Sulje kaikki portit ... JA tarkista Steppiä seuraavassa transitioehdossa, että kaikki portit ovat kiinni
Close all gates.... and check in following transition that ALL gates are closed*)

;
END_ACTION

ACTION ResetSFC_action:
(*Reset SFC*)
SFCReset:=TRUE;
END_ACTION
END_PROGRAM

(* POU OLD/PRG_ToColourSensor, SFC *)
PROGRAM PRG_ToColourSensor
VAR_INPUT
	bReset		: BOOL;	(*Reset program*)
	bExecute		: BOOL;	(*enable and run*)
END_VAR
VAR_OUTPUT
	bDone			: BOOL;
END_VAR
VAR

	tonMoveDelay	: TON;
	SFCReset		: BOOL;
	tMoveDelay	: TIME := T#4s;
END_VAR
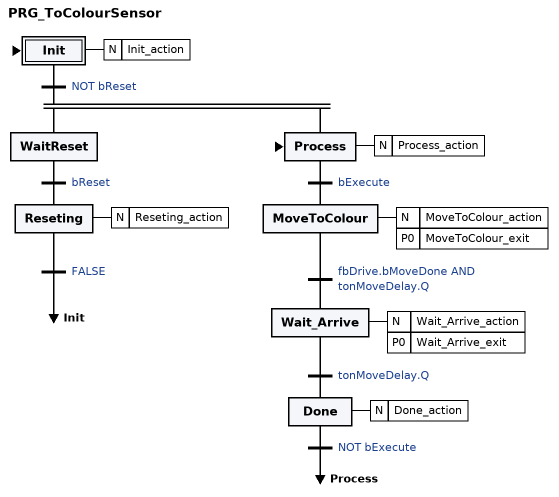
INITIAL_STEP Init:
	Init_action(N);
END_STEP
TRANSITION FROM Init TO (WaitReset, Process) := NOT bReset;
END_TRANSITION
STEP WaitReset:
END_STEP
TRANSITION FROM WaitReset TO Reseting := bReset;
END_TRANSITION
STEP Process:
	Process_action(N);
END_STEP
TRANSITION FROM Process TO MoveToColour := bExecute;
END_TRANSITION
STEP MoveToColour:
	MoveToColour_action(N);
	MoveToColour_exit(P0);
END_STEP
TRANSITION FROM MoveToColour TO Wait_Arrive := fbDrive.bMoveDone AND tonMoveDelay.Q;
END_TRANSITION
STEP Wait_Arrive:
	Wait_Arrive_action(N);
	Wait_Arrive_exit(P0);
END_STEP
TRANSITION FROM Wait_Arrive TO Done := tonMoveDelay.Q;
END_TRANSITION
STEP Done:
	Done_action(N);
END_STEP
TRANSITION FROM Done TO Process := NOT bExecute;
END_TRANSITION
STEP Reseting:
	Reseting_action(N);
END_STEP
TRANSITION FROM Reseting TO Init := FALSE;
END_TRANSITION

ACTION Init_action:
SFCReset := FALSE;
bDone := FALSE;
END_ACTION

ACTION Process_action:
bDone := FALSE;
END_ACTION

ACTION MoveToColour_action:
bDone := FALSE;

fbDrive(
	bEnable:= TRUE,
	bStart:= TRUE,
	wTarget:= GPOS_COLOR_SEN);

tonMoveDelay(IN:=TRUE , PT:= tMoveDelay);

(*
tonMoveDelay(IN:=TRUE , PT:= tMoveDelay);
*)
END_ACTION

ACTION MoveToColour_exit:
fbDrive(
	bStart:= FALSE);

tonMoveDelay(IN:=FALSE);
END_ACTION

ACTION Wait_Arrive_action:
tonMoveDelay(IN:=TRUE , PT:= tMoveDelay);
END_ACTION

ACTION Wait_Arrive_exit:
tonMoveDelay(IN:=FALSE);
END_ACTION

ACTION Done_action:
bDone := TRUE;
END_ACTION

ACTION Reseting_action:
SFCReset := TRUE;
END_ACTION
END_PROGRAM

(* POU OLD/PRG_ToColourSensor2, SFC *)
PROGRAM PRG_ToColourSensor2
VAR_INPUT
	bExecute: BOOL;
END_VAR
VAR_INPUT
	bDone: BOOL;
END_VAR
VAR
	tonMoveDelay	: TON;
	tonEjectDelay	: TON;
	tMoveDelay	: TIME := T#3s;
	tEjectorDelay	: TIME := T#3s;
END_VAR
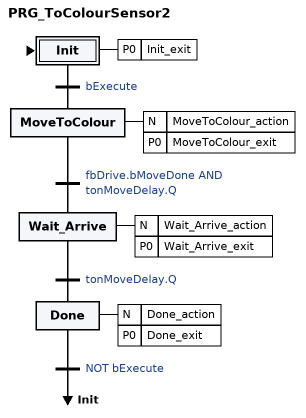
INITIAL_STEP Init:
	Init_exit(P0);
END_STEP
TRANSITION FROM Init TO MoveToColour := bExecute;
END_TRANSITION
STEP MoveToColour:
	MoveToColour_action(N);
	MoveToColour_exit(P0);
END_STEP
TRANSITION FROM MoveToColour TO Wait_Arrive := fbDrive.bMoveDone AND tonMoveDelay.Q;
END_TRANSITION
STEP Wait_Arrive:
	Wait_Arrive_action(N);
	Wait_Arrive_exit(P0);
END_STEP
TRANSITION FROM Wait_Arrive TO Done := tonMoveDelay.Q;
END_TRANSITION
STEP Done:
	Done_action(N);
	Done_exit(P0);
END_STEP
TRANSITION FROM Done TO Init := NOT bExecute;
END_TRANSITION

ACTION Init_exit:
bDone := FALSE;
END_ACTION

ACTION MoveToColour_action:
fbDrive(
	bEnable:= TRUE,
	bStart:= TRUE,
	wTarget:= GPOS_COLOR_SEN);

tonMoveDelay(IN:=TRUE , PT:= tMoveDelay);
END_ACTION

ACTION MoveToColour_exit:
fbDrive(
	bStart:= FALSE);
tonMoveDelay(IN:=FALSE);
END_ACTION

ACTION Wait_Arrive_action:
tonMoveDelay(IN:=TRUE , PT:= tMoveDelay);
END_ACTION

ACTION Wait_Arrive_exit:
tonMoveDelay(IN:=FALSE);
END_ACTION

ACTION Done_action:
bDone := TRUE;
END_ACTION

ACTION Done_exit:
bDone := FALSE;
END_ACTION
END_PROGRAM

(* POU OLD/FB_Lift2Old, SFC *)
FUNCTION_BLOCK FB_Lift2Old
VAR_INPUT
	bReset			 : BOOL;	(*Reset Request*)
	bEnable			 : BOOL;
	I_LimitUp 			 : BOOL;
	I_LimitLow 	        : BOOL;
	I_WaitingBallMetal : BOOL;

	(* ColourSensor *)
	I_SenColourYellow		:BOOL;	(*Colour sensor In1 - Yellow*)
	I_SenColourBlue		:BOOL;	(*Colour sensor In2 - Blue*)
	I_SenColourGreen		:BOOL;	(*Colour sensor In3 - Green*)
	I_SenColourRed		:BOOL;	(*Colour sensor In4 - Red*)

	(*SMEMA Handshake Inputs*)
	hiRdyToReceive_FromDS	: BOOL;
	hiBallAvail_FromUS		: BOOL;
END_VAR
VAR_OUTPUT
	bStopOK		: BOOL;
	bBallLoaded	: BOOL;
	bCurBallMetal	: BOOL;
	bCurrentBall 	: E_BallColour := NoColour;

	O_Ejector		:BOOL;

	(*SMEMA Handshake Outputs*)
	hoBallAvail_ToDS 			: BOOL;
	hoReadyToRecieve_ToUS		: BOOL;
END_VAR
VAR
	bBallRequested : BOOL := FALSE;
	fbTransferBall	:FB_TransferBall2;

	fbDelay		: FB_Wait;
	tonMoveDelay	: TON;
	tonSensorDelay	: TON;
	tTransferDelay: TIME := T#4s;
	tMoveDelay	: TIME := T#4s;
	tSensorDelay	: TIME := T#2s;
	bLocalReset	: BOOL;	(*Performs local reset*)
	SFCReset 	: BOOL;	(*Resets the execution of SFC to init once this SFCFlag is set true *)
END_VAR
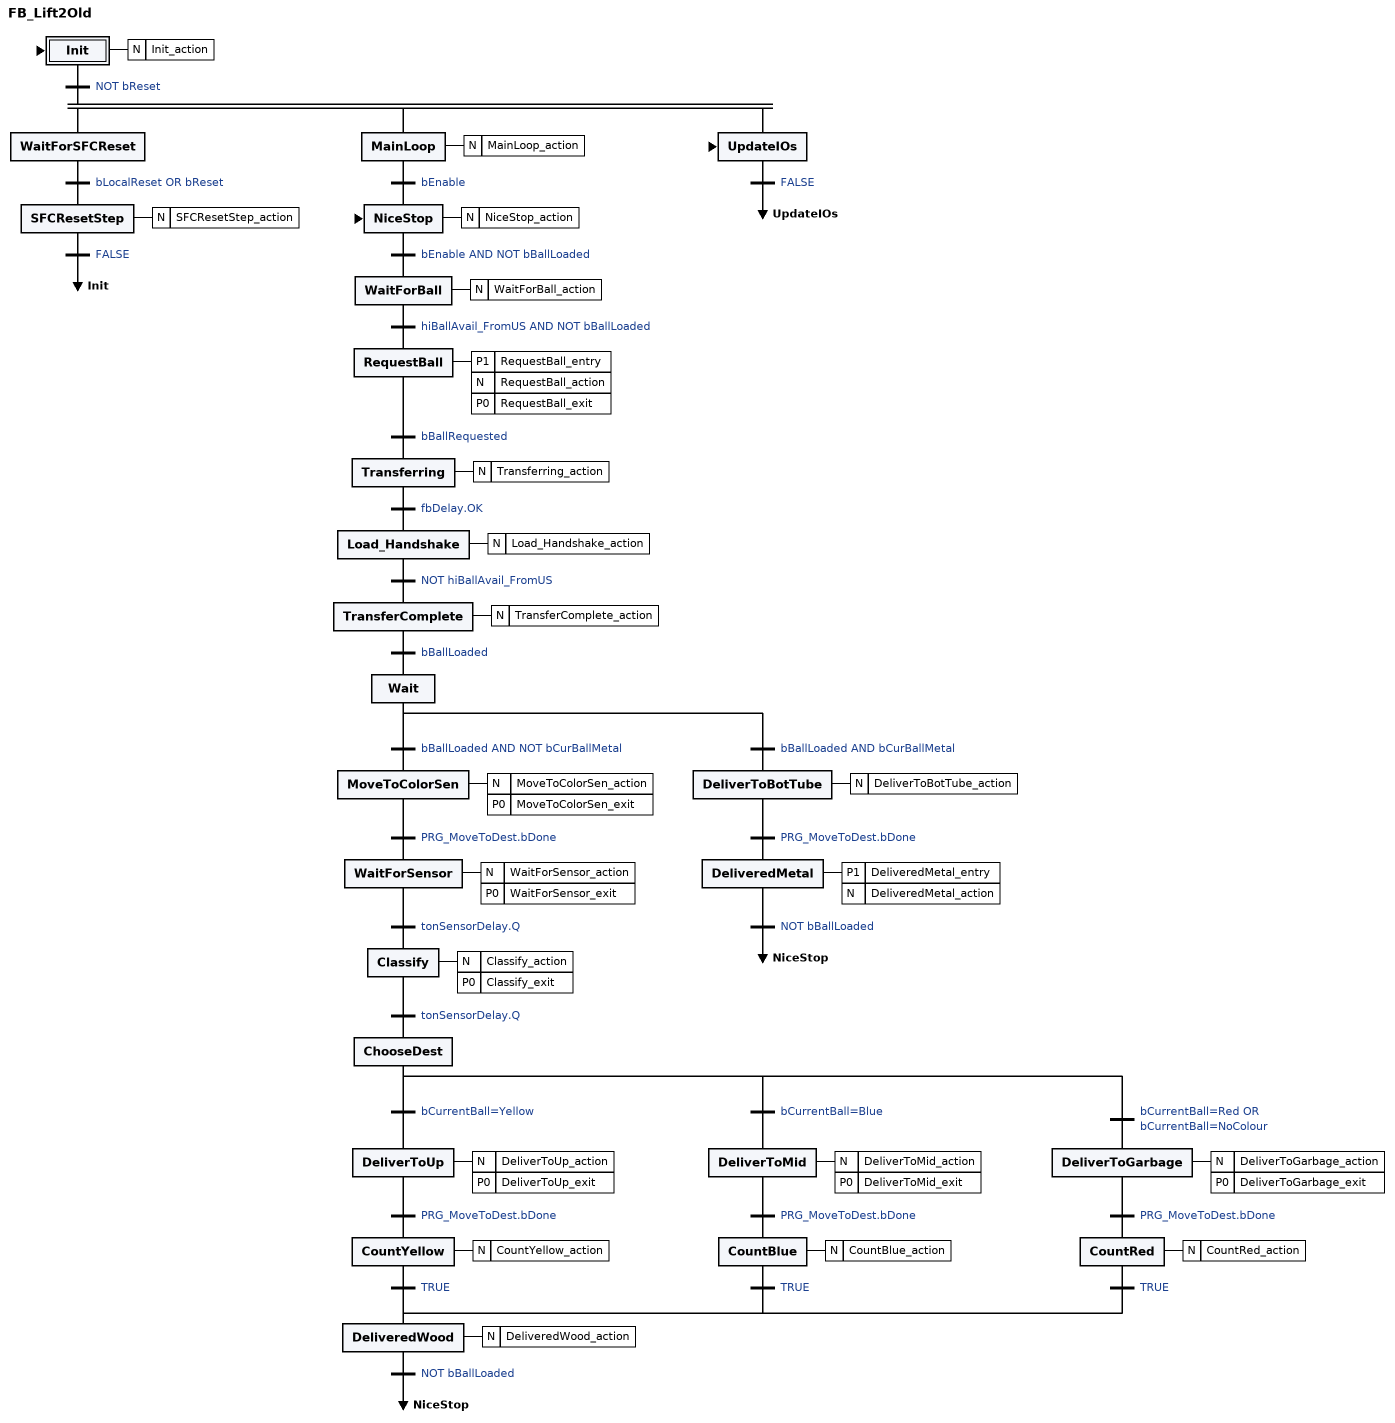
INITIAL_STEP Init:
	Init_action(N);
END_STEP
TRANSITION FROM Init TO (WaitForSFCReset, MainLoop, UpdateIOs) := NOT bReset;
END_TRANSITION
STEP WaitForSFCReset:
END_STEP
TRANSITION FROM WaitForSFCReset TO SFCResetStep := bLocalReset OR bReset;
END_TRANSITION
STEP MainLoop:
	MainLoop_action(N);
END_STEP
TRANSITION FROM MainLoop TO NiceStop := bEnable;
END_TRANSITION
STEP NiceStop:
	NiceStop_action(N);
END_STEP
TRANSITION FROM NiceStop TO WaitForBall := bEnable AND NOT bBallLoaded;
END_TRANSITION
STEP WaitForBall:
	WaitForBall_action(N);
END_STEP
TRANSITION FROM WaitForBall TO RequestBall := hiBallAvail_FromUS AND NOT bBallLoaded;
END_TRANSITION
STEP RequestBall:
	RequestBall_entry(P1);
	RequestBall_action(N);
	RequestBall_exit(P0);
END_STEP
TRANSITION FROM RequestBall TO Transferring := bBallRequested;
END_TRANSITION
STEP Transferring:
	Transferring_action(N);
END_STEP
TRANSITION FROM Transferring TO Load_Handshake := fbDelay.OK;
END_TRANSITION
STEP Load_Handshake:
	Load_Handshake_action(N);
END_STEP
TRANSITION FROM Load_Handshake TO TransferComplete := NOT hiBallAvail_FromUS;
END_TRANSITION
STEP TransferComplete:
	TransferComplete_action(N);
END_STEP
TRANSITION FROM TransferComplete TO Wait := bBallLoaded;
END_TRANSITION
STEP Wait:
END_STEP
TRANSITION FROM Wait TO MoveToColorSen := bBallLoaded AND NOT bCurBallMetal;
END_TRANSITION
TRANSITION FROM Wait TO DeliverToBotTube := bBallLoaded AND bCurBallMetal;
END_TRANSITION
STEP DeliverToBotTube:
	DeliverToBotTube_action(N);
END_STEP
TRANSITION FROM DeliverToBotTube TO DeliveredMetal := PRG_MoveToDest.bDone;
END_TRANSITION
STEP DeliveredMetal:
	DeliveredMetal_entry(P1);
	DeliveredMetal_action(N);
END_STEP
TRANSITION FROM DeliveredMetal TO NiceStop := NOT bBallLoaded;
END_TRANSITION
STEP MoveToColorSen:
	MoveToColorSen_action(N);
	MoveToColorSen_exit(P0);
END_STEP
TRANSITION FROM MoveToColorSen TO WaitForSensor := PRG_MoveToDest.bDone;
END_TRANSITION
STEP WaitForSensor:
	WaitForSensor_action(N);
	WaitForSensor_exit(P0);
END_STEP
TRANSITION FROM WaitForSensor TO Classify := tonSensorDelay.Q;
END_TRANSITION
STEP Classify:
	Classify_action(N);
	Classify_exit(P0);
END_STEP
TRANSITION FROM Classify TO ChooseDest := tonSensorDelay.Q;
END_TRANSITION
STEP ChooseDest:
END_STEP
TRANSITION FROM ChooseDest TO DeliverToUp := bCurrentBall=Yellow;
END_TRANSITION
TRANSITION FROM ChooseDest TO DeliverToMid := bCurrentBall=Blue;
END_TRANSITION
TRANSITION FROM ChooseDest TO DeliverToGarbage := bCurrentBall=Red OR bCurrentBall=NoColour;
END_TRANSITION
STEP DeliverToUp:
	DeliverToUp_action(N);
	DeliverToUp_exit(P0);
END_STEP
TRANSITION FROM DeliverToUp TO CountYellow := PRG_MoveToDest.bDone;
END_TRANSITION
STEP CountYellow:
	CountYellow_action(N);
END_STEP
TRANSITION FROM CountYellow TO DeliveredWood := TRUE;
END_TRANSITION
STEP DeliverToMid:
	DeliverToMid_action(N);
	DeliverToMid_exit(P0);
END_STEP
TRANSITION FROM DeliverToMid TO CountBlue := PRG_MoveToDest.bDone;
END_TRANSITION
STEP CountBlue:
	CountBlue_action(N);
END_STEP
TRANSITION FROM CountBlue TO DeliveredWood := TRUE;
END_TRANSITION
STEP DeliverToGarbage:
	DeliverToGarbage_action(N);
	DeliverToGarbage_exit(P0);
END_STEP
TRANSITION FROM DeliverToGarbage TO CountRed := PRG_MoveToDest.bDone;
END_TRANSITION
STEP CountRed:
	CountRed_action(N);
END_STEP
TRANSITION FROM CountRed TO DeliveredWood := TRUE;
END_TRANSITION
STEP DeliveredWood:
	DeliveredWood_action(N);
END_STEP
TRANSITION FROM DeliveredWood TO NiceStop := NOT bBallLoaded;
END_TRANSITION
STEP UpdateIOs:
END_STEP
TRANSITION FROM UpdateIOs TO UpdateIOs := FALSE;
END_TRANSITION
STEP SFCResetStep:
	SFCResetStep_action(N);
END_STEP
TRANSITION FROM SFCResetStep TO Init := FALSE;
END_TRANSITION

ACTION Init_action:
SFCReset := FALSE;
bLocalReset	:= FALSE;
END_ACTION

ACTION MainLoop_action:
hoBallAvail_ToDS			  := FALSE;
hoReadyToRecieve_ToUS := FALSE;
END_ACTION

ACTION NiceStop_action:
bStopOK	  	:= TRUE;
bCurrentBall	:= NoColour;
END_ACTION

ACTION WaitForBall_action:
bBallLoaded := FALSE;
hoReadyToRecieve_ToUS := TRUE;
END_ACTION

ACTION RequestBall_entry:
bStopOK := FALSE;
END_ACTION

ACTION RequestBall_action:
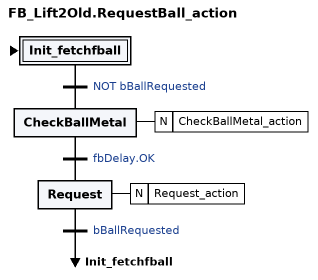
INITIAL_STEP Init_fetchfball:
END_STEP
TRANSITION FROM Init_fetchfball TO CheckBallMetal := NOT bBallRequested;
END_TRANSITION
STEP CheckBallMetal:
	CheckBallMetal_action(N);
END_STEP
TRANSITION FROM CheckBallMetal TO Request := fbDelay.OK;
END_TRANSITION
STEP Request:
	Request_action(N);
END_STEP
TRANSITION FROM Request TO Init_fetchfball := bBallRequested;
END_TRANSITION

ACTION CheckBallMetal_action:
bCurBallMetal	 := I_WaitingBallMetal;
fbDelay(IN_TIME:=T#2s);
END_ACTION

ACTION Request_action:
hoReadyToRecieve_ToUS := TRUE;
bBallRequested := TRUE;
END_ACTION
END_ACTION

ACTION RequestBall_exit:
bBallRequested := FALSE;
END_ACTION

ACTION Transferring_action:
fbDelay(IN_TIME:=tTransferDelay);
END_ACTION

ACTION Load_Handshake_action:
hoReadyToRecieve_ToUS := FALSE;
END_ACTION

ACTION TransferComplete_action:
bBallLoaded := TRUE;
END_ACTION

ACTION DeliverToBotTube_action:
PRG_MoveToDest(bExecute:= TRUE, wTarget:= GPOS_PIPE_LOW, bDone:= );
END_ACTION

ACTION DeliveredMetal_entry:
bBallLoaded := FALSE;
PRG_MoveToDest( bExecute:=FALSE);
END_ACTION

ACTION DeliveredMetal_action:
bBallLoaded := FALSE;
CountBallsSortedMetal := CountBallsSortedMetal + 1;
arrCountBallsOnTubes[1] := arrCountBallsOnTubes[1] + 1;
END_ACTION

ACTION MoveToColorSen_action:
PRG_MoveToDest(bExecute:= TRUE, wTarget:= GPOS_COLOR_SEN, bDone:= );
END_ACTION

ACTION MoveToColorSen_exit:
PRG_MoveToDest( bExecute:=FALSE);
END_ACTION

ACTION WaitForSensor_action:
tonSensorDelay(IN:=TRUE , PT:= tSensorDelay);
END_ACTION

ACTION WaitForSensor_exit:
tonSensorDelay(IN:=FALSE);
END_ACTION

ACTION Classify_action:
tonSensorDelay(IN:=TRUE , PT:= tSensorDelay);
IF I_SenColourYellow THEN
	bCurrentBall := Yellow;
ELSIF  I_SenColourBlue THEN
	bCurrentBall := Blue;
ELSIF  I_SenColourRed THEN
	bCurrentBall := Red;
ELSE
	bCurrentBall := NoColour;
END_IF
END_ACTION

ACTION Classify_exit:
tonSensorDelay(IN:=FALSE);
END_ACTION

ACTION DeliverToUp_action:
PRG_MoveToDest(bExecute:= TRUE , wTarget:= GPOS_PIPE_UP, bDone:= );
END_ACTION

ACTION DeliverToUp_exit:
PRG_MoveToDest(bExecute:= FALSE);
END_ACTION

ACTION CountYellow_action:
CountBallsSortedYellow := CountBallsSortedYellow + 1;
CountBallsSortedWooden := CountBallsSortedWooden + 1;
arrCountBallsOnTubes[3] := arrCountBallsOnTubes[3] + 1;
END_ACTION

ACTION DeliverToMid_action:
PRG_MoveToDest(bExecute:= TRUE , wTarget:= GPOS_PIPE_MID, bDone:= );
END_ACTION

ACTION DeliverToMid_exit:
PRG_MoveToDest(bExecute:= FALSE);
END_ACTION

ACTION CountBlue_action:
CountBallsSortedBlue := CountBallsSortedBlue + 1;
CountBallsSortedWooden := CountBallsSortedWooden + 1;
arrCountBallsOnTubes[2] := arrCountBallsOnTubes[2] + 1;
END_ACTION

ACTION DeliverToGarbage_action:
PRG_MoveToDest(bExecute:= TRUE , wTarget:= GPOS_GARBAGE, bDone:= );
END_ACTION

ACTION DeliverToGarbage_exit:
PRG_MoveToDest(bExecute:= FALSE);
END_ACTION

ACTION CountRed_action:
CountBallsSortedRed := CountBallsSortedRed + 1;
CountBallsSortedGarbage := CountBallsSortedGarbage + 1;
CountBallsSortedWooden := CountBallsSortedWooden + 1;
arrCountBallsOnTubes[4] := arrCountBallsOnTubes[4] + 1;
END_ACTION

ACTION DeliveredWood_action:
bBallLoaded := FALSE;
bCurrentBall := NoColour;
END_ACTION

ACTION SFCResetStep_action:
SFCReset := TRUE;
END_ACTION
END_FUNCTION_BLOCK

(* POU OLD/FB_TransferBall2, ST *)
FUNCTION_BLOCK FB_TransferBall2
VAR_INPUT
	bExecute			: BOOL;	(*enable and run*)
	bBallToTransfer 	: E_BallColour;
END_VAR
VAR_OUTPUT
	bDone			: BOOL := FALSE;
END_VAR
VAR
	tonMoveDelay	: TON;
	tonEjectDelay	: TON;
	tMoveDelay	: TIME := T#1s;
	tEjectorDelay	: TIME := T#1s;
END_VAR
IF bExecute THEN
	CASE bBallToTransfer OF
		Yellow:
			PRG_MoveToDest(bExecute:= TRUE , wTarget:= GPOS_PIPE_UP, bDone:= );
			bDone	:= FALSE;
		Blue:
			PRG_MoveToDest(bExecute:= TRUE , wTarget:= GPOS_PIPE_MID, bDone:= );
				bDone	:= FALSE;
		Red, NoColour:
			PRG_MoveToDest(bExecute:= TRUE , wTarget:= GPOS_GARBAGE, bDone:= );
				bDone	:= FALSE;
	ELSE
		PRG_MoveToDest(bExecute:=FALSE);
		bDone	:= FALSE;
	END_CASE

	IF PRG_MoveToDest.bDone THEN
		PRG_MoveToDest(bExecute:=FALSE);
		bDone	:= TRUE;
	END_IF

ELSE
	bDone := FALSE;
END_IF
END_FUNCTION_BLOCK

(* POU OLD/FB_Lift_Old, SFC *)
FUNCTION_BLOCK FB_Lift_Old
VAR_INPUT
	bReset			 : BOOL;	(*Reset Request*)
	bEnable			 : BOOL;
	I_LimitUp 			 : BOOL;
	I_LimitLow 	        : BOOL;
	I_WaitingBallMetal : BOOL;

	(* ColourSensor *)
	I_SenColourYellow		:BOOL;	(*Colour sensor In1 - Yellow*)
	I_SenColourBlue		:BOOL;	(*Colour sensor In2 - Blue*)
	I_SenColourGreen		:BOOL;	(*Colour sensor In3 - Green*)
	I_SenColourRed		:BOOL;	(*Colour sensor In4 - Red*)

	(*SMEMA Handshake Inputs*)
	hiRdyToReceive_FromDS	: BOOL;
	hiBallAvail_FromUS		: BOOL;
END_VAR
VAR_OUTPUT
	bStopOK		: BOOL;
	bBallLoaded	: BOOL;
	bCurBallMetal	: BOOL;
	bCurrentBall 	: E_BallColour := NoColour;

	O_Ejector		:BOOL;

	(*SMEMA Handshake Outputs*)
	hoBallAvail_ToDS 			: BOOL;
	hoReadyToRecieve_ToUS		: BOOL;
END_VAR
VAR
	bBallRequested : BOOL := FALSE;
	fbTransferBall	:FB_TransferBall2;

	fbDelay		: FB_Wait;
	tonMoveDelay	: TON;
	tonSensorDelay	: TON;
	tTransferDelay: TIME := T#4s;
	tMoveDelay	: TIME := T#4s;
	tSensorDelay	: TIME := T#2s;
	bLocalReset	: BOOL;	(*Performs local reset*)
	SFCReset 	: BOOL;	(*Resets the execution of SFC to init once this SFCFlag is set true *)
END_VAR
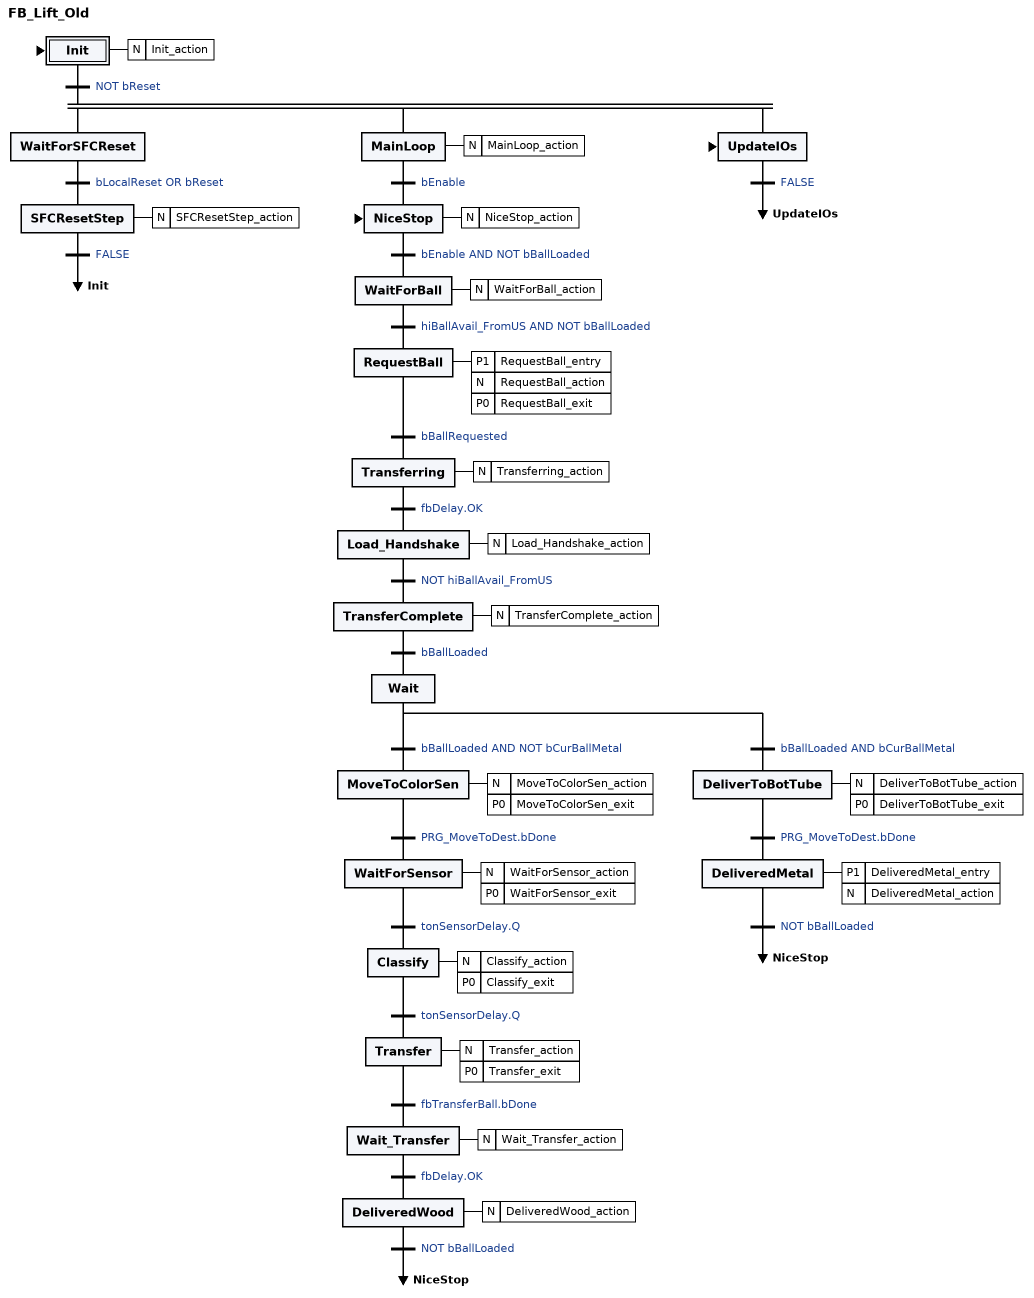
INITIAL_STEP Init:
	Init_action(N);
END_STEP
TRANSITION FROM Init TO (WaitForSFCReset, MainLoop, UpdateIOs) := NOT bReset;
END_TRANSITION
STEP WaitForSFCReset:
END_STEP
TRANSITION FROM WaitForSFCReset TO SFCResetStep := bLocalReset OR bReset;
END_TRANSITION
STEP MainLoop:
	MainLoop_action(N);
END_STEP
TRANSITION FROM MainLoop TO NiceStop := bEnable;
END_TRANSITION
STEP NiceStop:
	NiceStop_action(N);
END_STEP
TRANSITION FROM NiceStop TO WaitForBall := bEnable AND NOT bBallLoaded;
END_TRANSITION
STEP WaitForBall:
	WaitForBall_action(N);
END_STEP
TRANSITION FROM WaitForBall TO RequestBall := hiBallAvail_FromUS AND NOT bBallLoaded;
END_TRANSITION
STEP RequestBall:
	RequestBall_entry(P1);
	RequestBall_action(N);
	RequestBall_exit(P0);
END_STEP
TRANSITION FROM RequestBall TO Transferring := bBallRequested;
END_TRANSITION
STEP Transferring:
	Transferring_action(N);
END_STEP
TRANSITION FROM Transferring TO Load_Handshake := fbDelay.OK;
END_TRANSITION
STEP Load_Handshake:
	Load_Handshake_action(N);
END_STEP
TRANSITION FROM Load_Handshake TO TransferComplete := NOT hiBallAvail_FromUS;
END_TRANSITION
STEP TransferComplete:
	TransferComplete_action(N);
END_STEP
TRANSITION FROM TransferComplete TO Wait := bBallLoaded;
END_TRANSITION
STEP Wait:
END_STEP
TRANSITION FROM Wait TO MoveToColorSen := bBallLoaded AND NOT bCurBallMetal;
END_TRANSITION
TRANSITION FROM Wait TO DeliverToBotTube := bBallLoaded AND bCurBallMetal;
END_TRANSITION
STEP DeliverToBotTube:
	DeliverToBotTube_action(N);
	DeliverToBotTube_exit(P0);
END_STEP
TRANSITION FROM DeliverToBotTube TO DeliveredMetal := PRG_MoveToDest.bDone;
END_TRANSITION
STEP DeliveredMetal:
	DeliveredMetal_entry(P1);
	DeliveredMetal_action(N);
END_STEP
TRANSITION FROM DeliveredMetal TO NiceStop := NOT bBallLoaded;
END_TRANSITION
STEP MoveToColorSen:
	MoveToColorSen_action(N);
	MoveToColorSen_exit(P0);
END_STEP
TRANSITION FROM MoveToColorSen TO WaitForSensor := PRG_MoveToDest.bDone;
END_TRANSITION
STEP WaitForSensor:
	WaitForSensor_action(N);
	WaitForSensor_exit(P0);
END_STEP
TRANSITION FROM WaitForSensor TO Classify := tonSensorDelay.Q;
END_TRANSITION
STEP Classify:
	Classify_action(N);
	Classify_exit(P0);
END_STEP
TRANSITION FROM Classify TO Transfer := tonSensorDelay.Q;
END_TRANSITION
STEP Transfer:
	Transfer_action(N);
	Transfer_exit(P0);
END_STEP
TRANSITION FROM Transfer TO Wait_Transfer := fbTransferBall.bDone;
END_TRANSITION
STEP Wait_Transfer:
	Wait_Transfer_action(N);
END_STEP
TRANSITION FROM Wait_Transfer TO DeliveredWood := fbDelay.OK;
END_TRANSITION
STEP DeliveredWood:
	DeliveredWood_action(N);
END_STEP
TRANSITION FROM DeliveredWood TO NiceStop := NOT bBallLoaded;
END_TRANSITION
STEP UpdateIOs:
END_STEP
TRANSITION FROM UpdateIOs TO UpdateIOs := FALSE;
END_TRANSITION
STEP SFCResetStep:
	SFCResetStep_action(N);
END_STEP
TRANSITION FROM SFCResetStep TO Init := FALSE;
END_TRANSITION

ACTION Init_action:
SFCReset := FALSE;
bLocalReset	:= FALSE;
END_ACTION

ACTION MainLoop_action:
hoBallAvail_ToDS			  := FALSE;
hoReadyToRecieve_ToUS := FALSE;
END_ACTION

ACTION NiceStop_action:
bStopOK	  	:= TRUE;
bCurrentBall	:= NoColour;
END_ACTION

ACTION WaitForBall_action:
bBallLoaded := FALSE;
hoReadyToRecieve_ToUS := TRUE;
END_ACTION

ACTION RequestBall_entry:
bStopOK := FALSE;
END_ACTION

ACTION RequestBall_action:
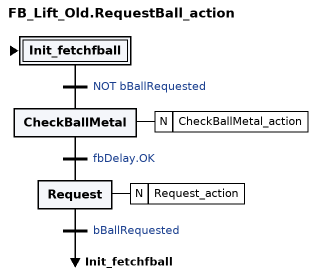
INITIAL_STEP Init_fetchfball:
END_STEP
TRANSITION FROM Init_fetchfball TO CheckBallMetal := NOT bBallRequested;
END_TRANSITION
STEP CheckBallMetal:
	CheckBallMetal_action(N);
END_STEP
TRANSITION FROM CheckBallMetal TO Request := fbDelay.OK;
END_TRANSITION
STEP Request:
	Request_action(N);
END_STEP
TRANSITION FROM Request TO Init_fetchfball := bBallRequested;
END_TRANSITION

ACTION CheckBallMetal_action:
bCurBallMetal	 := I_WaitingBallMetal;
fbDelay(IN_TIME:=T#2s);
END_ACTION

ACTION Request_action:
hoReadyToRecieve_ToUS := TRUE;
bBallRequested := TRUE;
END_ACTION
END_ACTION

ACTION RequestBall_exit:
bBallRequested := FALSE;
END_ACTION

ACTION Transferring_action:
fbDelay(IN_TIME:=tTransferDelay);
END_ACTION

ACTION Load_Handshake_action:
hoReadyToRecieve_ToUS := FALSE;
END_ACTION

ACTION TransferComplete_action:
bBallLoaded := TRUE;
END_ACTION

ACTION DeliverToBotTube_action:
PRG_MoveToDest(bExecute:= TRUE, wTarget:= GPOS_PIPE_LOW, bDone:= );
END_ACTION

ACTION DeliverToBotTube_exit:
PRG_MoveToDest( bExecute:=FALSE);
END_ACTION

ACTION DeliveredMetal_entry:
bBallLoaded := FALSE;
PRG_DeliverToLow(bReset:=FALSE , bExecute:=FALSE ,  bDone=> );
END_ACTION

ACTION DeliveredMetal_action:
bBallLoaded := FALSE;
END_ACTION

ACTION MoveToColorSen_action:
PRG_MoveToDest(bExecute:= TRUE, wTarget:= GPOS_COLOR_SEN, bDone:= );
END_ACTION

ACTION MoveToColorSen_exit:
PRG_MoveToDest( bExecute:=FALSE);
END_ACTION

ACTION WaitForSensor_action:
tonSensorDelay(IN:=TRUE , PT:= tSensorDelay);
END_ACTION

ACTION WaitForSensor_exit:
tonSensorDelay(IN:=FALSE);
END_ACTION

ACTION Classify_action:
tonSensorDelay(IN:=TRUE , PT:= tSensorDelay);
IF I_SenColourYellow THEN
	bCurrentBall := Yellow;
ELSIF  I_SenColourBlue THEN
	bCurrentBall := Blue;
ELSIF  I_SenColourRed THEN
	bCurrentBall := Red;
ELSE
	bCurrentBall := NoColour;
END_IF
END_ACTION

ACTION Classify_exit:
tonSensorDelay(IN:=FALSE);
END_ACTION

ACTION Transfer_action:
fbTransferBall(bExecute:= TRUE , bBallToTransfer:= bCurrentBall, bDone=> );
END_ACTION

ACTION Transfer_exit:
fbTransferBall(bExecute:= FALSE);
END_ACTION

ACTION Wait_Transfer_action:
fbDelay(IN_TIME:=tMoveDelay);
END_ACTION

ACTION DeliveredWood_action:
bBallLoaded := FALSE;
bCurrentBall := NoColour;
END_ACTION

ACTION SFCResetStep_action:
SFCReset := TRUE;
END_ACTION
END_FUNCTION_BLOCK

(* POU FBs/FB_StateModel_ST, ST *)
FUNCTION_BLOCK FB_StateModel_ST
(*PackML State model implementation. Slightly modified implementation.
Author: 	Niko Siltala, niko.siltala@tut.fi
Date: 	2016-01-29
*)
VAR_INPUT
	bResetFB	: BOOL;		(*Resets whole FB*)
	eModeReq	: E_ModeCtrl;	(*Requested mode*)
	wIgnoreState	: DWORD;	(*Ignoring states. See bit from E_State definition. Aborting = bit0*)
	bSC			: BOOL;		(*Step Completed acknoledgement*)
	bAbort		: BOOL;		(*Abortting signal = EmergencyStop*)
	bClear		: BOOL;		(*Clear signal*)
	bReset		: BOOL;		(*Reseting signal*)
	bStart		: BOOL;		(*Start signal*)
	bHold		: BOOL;		(*Hold signal*)
	bUn_Hold	: BOOL;		(*Un-Hold signal*)
	bSuspend	: BOOL;		(*Suspend signal*)
	bUn_Suspend	: BOOL;		(*Un-Suspend signal*)
	bStop		: BOOL;		(*Stop signal*)
	bComplete	: BOOL;		(*Complete signal*)
	bAck_Completed	: BOOL;	(*Acknoledgement for Complete signal*)
END_VAR
VAR_OUTPUT
	eMode	: E_ModeCtrl;	(*Current mode*)
	eState	: E_State;	(*Current state*)
END_VAR
VAR
	RTrig_bSC	: R_TRIG; 	(*Rising trigger for State Completed*)
	RTrig_StateChange	: R_TRIG; 	(*Rising trigger for State signal*)
	bResetLocal		: BOOL:=FALSE;	(*Paikallinen Reset*)
	bInitDone	: BOOL;		(*Initialisation*)
END_VAR
IF bResetFB THEN	(*Reseting FB*)
	bInitDone := FALSE;
END_IF;

(*Initialisation*)
IF NOT bInitDone THEN
	eState:= eSt_Aborting;
	bInitDone:=TRUE;
END_IF;

(*Rising triggers monitor*)
RTrig_bSC(CLK:=bSC , Q=> );

(*Abort signal interrupt*)
IF bAbort AND (eState > eSt_Clearing) THEN
	eState:=eSt_Aborting;
END_IF;

(*Stop signal interrupt*)
IF bStop AND (eState > eSt_Stopping) THEN
	eState:=eSt_Stopping;
END_IF;


(*Main case structure*)
CASE eState OF
eSt_Aborting:
	IF bSC THEN
		eState:=eSt_Aborted;
	END_IF;

eSt_Aborted:
	eMode:=eModeReq;	(*Change Mode*)
	IF bClear AND NOT bAbort THEN
		eState:=eSt_Clearing;
	END_IF;

eSt_Clearing:
	IF bAbort THEN
		eState:=eSt_Aborting;
	ELSIF bSC THEN
		eState:=eSt_Stopped;
		RTrig_StateChange(CLK:=bReset , Q=> );
	END_IF;

eSt_Stopping:
	IF bSC THEN
		eState:=eSt_Stopped;
		RTrig_StateChange(CLK:=bReset , Q=> );
	END_IF;

eSt_Stopped:
	eMode:=eModeReq;	(*Change Mode*)
	RTrig_StateChange(CLK:=bReset , Q=> );
(*	ELSIF NOT bStop AND (RTrig_StateChange.Q OR (wIgnoreState.5 AND bStart) ) THEN*)
	IF NOT bStop THEN	(*Stop signal is not active.*)
		IF wIgnoreState.5 AND bStart THEN	(*Reset state is ignored and going directly to start *)
			eState:=eSt_Idle;
		ELSIF RTrig_StateChange.Q THEN 	(*Rising edge for reset*)
			eState:=eSt_Resetting;
		END_IF;
	END_IF;

eSt_Resetting:
	IF bSC OR wIgnoreState.5 THEN
		eState:=eSt_Idle;
	END_IF;

eSt_Idle:
	eMode:=eModeReq;	(*Change Mode*)
	IF bStart OR wIgnoreState.6 THEN
		eState:=eSt_Starting;
	END_IF;

eSt_Starting:
	IF bSC OR wIgnoreState.7 THEN
		eState:=eSt_Execute;
	END_IF;

eSt_Execute:
	IF bComplete THEN
		eState:=eSt_Completing;
	ELSIF bHold THEN
		eState:=eSt_Holding;
	ELSIF bSuspend THEN
		eState:=eSt_Suspending;
	END_IF;

eSt_Holding:
	IF bSC THEN
		eState:=eSt_Held;
	END_IF;

eSt_Held:
	IF bUn_Hold AND NOT bHold THEN
		eState:=eSt_UnHolding;
	END_IF;

eSt_UnHolding:
	IF bSC THEN
		eState:=eSt_Execute;
	END_IF;

eSt_Suspending:
	IF bSC THEN
		eState:=eSt_Suspended;
	END_IF;

eSt_Suspended:
	IF bUn_Suspend AND NOT bSuspend THEN
		eState:=eSt_Unsuspending;
	END_IF;

eSt_Unsuspending:
	IF bSC THEN
		eState:=eSt_Execute;
	END_IF;

eSt_Completing:
	IF RTrig_bSC.Q THEN
		eState:=eSt_Completed;
	END_IF;

eSt_Completed:
	IF bAck_Completed THEN
		eState:=eSt_Resetting;
	END_IF;

ELSE
	(*Default error handler. Undefined state set*)
	eState:=eSt_Aborting;
END_CASE;
END_FUNCTION_BLOCK

(* POU OLD/FB_TransferBall, ST *)
FUNCTION_BLOCK FB_TransferBall
VAR_INPUT
	bExecute			: BOOL;	(*enable and run*)
	bBallToTransfer 	: E_BallColour;
END_VAR
VAR_OUTPUT
	bDone			: BOOL;
	bActDone		: BOOL := FALSE;
END_VAR
VAR
	tonMoveDelay	: TON;
	tonEjectDelay	: TON;
	tMoveDelay	: TIME := T#1s;
	tEjectorDelay	: TIME := T#1s;
END_VAR
IF bExecute THEN
	CASE bBallToTransfer OF
		Yellow:
			PRG_DeliverToUp2( bExecute:= TRUE , bDone=> );
				bDone	:= FALSE;
				IF PRG_DeliverToUp2.bDone THEN
					PRG_DeliverToUp2(bExecute:=FALSE);
					bDone	:= TRUE;
				END_IF
		Blue:
			PRG_DeliverToMid2( bExecute:= TRUE, bDone=> );
				bDone	:= FALSE;
				IF PRG_DeliverToMid2.bDone THEN
					PRG_DeliverToMid2(bExecute:=FALSE);
					bDone	:= TRUE;
				END_IF
		Red, NoColour:
			PRG_DeliverToGarbage2( bExecute:= TRUE, bDone=> );
				bDone	:= FALSE;
				IF PRG_DeliverToGarbage2.bDone THEN
					PRG_DeliverToGarbage2( bExecute:=FALSE);
					bDone	:= TRUE;
				END_IF
	ELSE
		PRG_DeliverToMid2(bExecute:=FALSE);
		PRG_DeliverToUp2(bExecute:=FALSE);
		PRG_DeliverToGarbage2( bExecute:=FALSE);
		bDone	:= FALSE;
	END_CASE
ELSE
	bDone := FALSE;
END_IF
END_FUNCTION_BLOCK

(* Visualisation FBs_Visu/FB_DRIVEMOVEMENTORIG
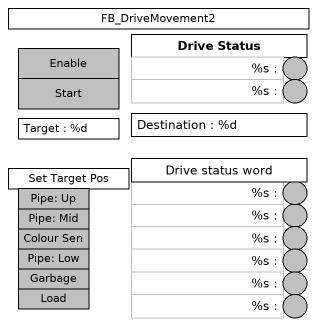
rectangle at (0,30)-(121,311): invisible if NOT .bManualMode
rectangle at (0,0)-(301,21): text "FB_DriveMovement2"
rectangle at (10,110)-(111,131): text "Target : %d"; shows $FB$.wTarget
rectangle at (10,40)-(111,71): text "Enable"; alarm colour if $FB$.bEnable; toggles $FB$.bEnable
rectangle at (10,70)-(111,101): text "Start"; alarm colour if $FB$.bStart; toggles $FB$.bStart
rectangle at (10,280)-(81,301): text "Load"; alarm colour if $FB$.wTarget = .GPOS_LOADING; runs INTERN ASSIGN $FB$.wTarget:=(GPOS_LOADING)
rectangle at (10,260)-(81,281): text "Garbage"; alarm colour if $FB$.wTarget = .GPOS_GARBAGE; runs INTERN ASSIGN $FB$.wTarget:=(GPOS_GARBAGE)
rectangle at (0,160)-(121,181): text "Set Target Pos"
rectangle at (10,240)-(81,261): text "Pipe: Low"; alarm colour if $FB$.wTarget = .GPOS_PIPE_LOW; runs INTERN ASSIGN $FB$.wTarget:=(GPOS_PIPE_LOW)
rectangle at (10,220)-(81,241): text "Colour Sen"; alarm colour if $FB$.wTarget = .GPOS_COLOR_SEN; runs INTERN ASSIGN $FB$.wTarget:=(GPOS_COLOR_SEN)
rectangle at (10,200)-(81,221): text "Pipe: Mid"; alarm colour if $FB$.wTarget = .GPOS_PIPE_MID; runs INTERN ASSIGN $FB$.wTarget:=(GPOS_PIPE_MID)
rectangle at (10,180)-(81,201): text "Pipe: Up"; alarm colour if $FB$.wTarget = .GPOS_PIPE_UP; runs INTERN ASSIGN $FB$.wTarget:=(GPOS_PIPE_UP)
embedded screen at (123,26)-(299,310): FB_VC_Drive_Status
*)

(* Visualisation FBs_Visu/FB_VC_Drive_Status
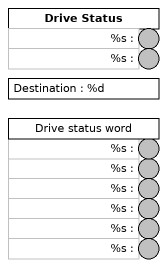
embedded screen at (0,150)-(151,171): VC_BOOLEANSTATUS
rectangle at (0,0)-(151,21): text "Drive Status"
embedded screen at (0,170)-(151,191): VC_BOOLEANSTATUS
embedded screen at (0,130)-(151,151): VC_BOOLEANSTATUS
embedded screen at (0,190)-(151,211): VC_BOOLEANSTATUS
embedded screen at (0,210)-(151,231): VC_BOOLEANSTATUS
embedded screen at (0,230)-(151,251): VC_BOOLEANSTATUS
rectangle at (0,70)-(151,91): text "Destination : %d"; shows $FB$.wDestination
rectangle at (0,110)-(151,131): text "Drive status word"
embedded screen at (0,20)-(151,41): VC_BOOLEANSTATUS
embedded screen at (0,40)-(151,61): VC_BOOLEANSTATUS
*)

(* Visualisation FBs_Visu/FB_VC_DRIVECONTROLS
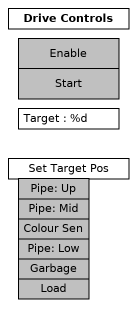
rectangle at (0,19)-(121,300): invisible if NOT .bManualMode
rectangle at (10,99)-(111,120): text "Target : %d"; shows $FB$.wTarget
rectangle at (10,29)-(111,60): text "Enable"; alarm colour if $FB$.bEnable; toggles $FB$.bEnable
rectangle at (10,59)-(111,90): text "Start"; alarm colour if $FB$.bStart; toggles $FB$.bStart
rectangle at (10,269)-(81,290): text "Load"; alarm colour if $FB$.wTarget = .GPOS_LOADING; runs INTERN ASSIGN $FB$.wTarget:=(GPOS_LOADING)
rectangle at (10,249)-(81,270): text "Garbage"; alarm colour if $FB$.wTarget = .GPOS_GARBAGE; runs INTERN ASSIGN $FB$.wTarget:=(GPOS_GARBAGE)
rectangle at (0,149)-(121,170): text "Set Target Pos"
rectangle at (10,229)-(81,250): text "Pipe: Low"; alarm colour if $FB$.wTarget = .GPOS_PIPE_LOW; runs INTERN ASSIGN $FB$.wTarget:=(GPOS_PIPE_LOW)
rectangle at (10,209)-(81,230): text "Colour Sen"; alarm colour if $FB$.wTarget = .GPOS_COLOR_SEN; runs INTERN ASSIGN $FB$.wTarget:=(GPOS_COLOR_SEN)
rectangle at (10,189)-(81,210): text "Pipe: Mid"; alarm colour if $FB$.wTarget = .GPOS_PIPE_MID; runs INTERN ASSIGN $FB$.wTarget:=(GPOS_PIPE_MID)
rectangle at (10,169)-(81,190): text "Pipe: Up"; alarm colour if $FB$.wTarget = .GPOS_PIPE_UP; runs INTERN ASSIGN $FB$.wTarget:=(GPOS_PIPE_UP)
rectangle at (0,-1)-(121,20): text "Drive Controls"
*)

(* Visualisation V_DRIVE
embedded screen at (0,0)-(401,311): FB_DriveMovement2
*)

(* Visualisation V_MAIN
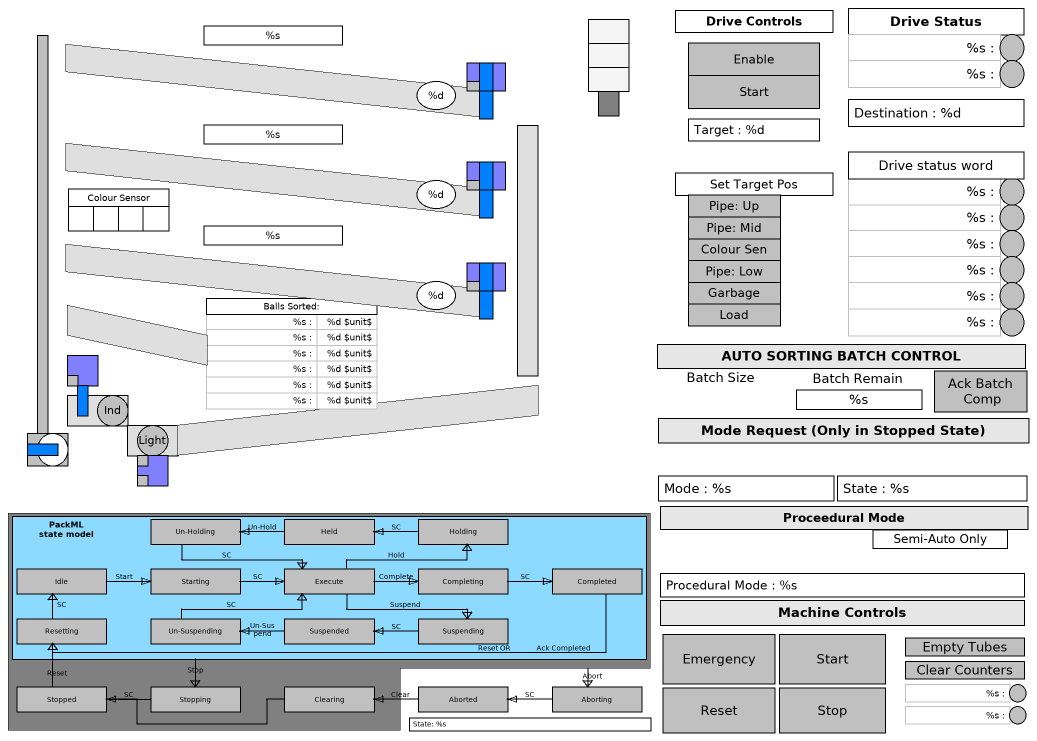
embedded screen at (60,340)-(531,471): VC_Graph_Sorter
embedded screen at (20,20)-(61,451): VC_Graph_Lift
embedded screen at (199,283)-(370,394): VC_Graph_Counters
embedded screen at (1,498)-(644,716): VC_PackMLStates
embedded screen at (46,-17)-(549,104): VC_PIPE
embedded screen at (46,82)-(549,203): VC_PIPE
embedded screen at (46,183)-(549,304): VC_PIPE
embedded screen at (61,172)-(162,216): VC_ColourSensor
embedded screen at (653,585)-(1019,718): VC_PANEL_MACHINECONTROL
embedded screen at (581,4)-(622,101): VC_Beacon
embedded screen at (841,-7)-(1017,321): FB_VC_Drive_Status
embedded screen at (668,-5)-(826,322): FB_VC_DriveControls
embedded screen at (653,491)-(1021,582): VC_PANEL_PROCMODESELECT
embedded screen at (651,403)-(1022,486): VC_PANEL_MODESELECTOR
embedded screen at (650,329)-(1020,397): VC_PANEL_BATCHCONTROL
2 more shapes without text or variables
*)

(* Visualisation Simulator/Components/VC_Beacon
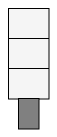
rectangle at (0,0)-(41,31): alarm colour if $red$
rectangle at (0,30)-(41,61): alarm colour if $yellow$
rectangle at (0,60)-(41,91): alarm colour if $green$
1 more shapes without text or variables
*)

(* Visualisation Components/VC_BOOLEANSTATUS
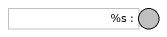
rectangle at (0,0)-(131,21): text "%s :"; shows $Name$
ellipse at (130,0)-(151,21): alarm colour if $bFlag$
*)

(* Visualisation Components/VC_ColourSensor
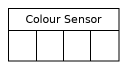
rectangle at (0,2)-(111,25): text "Colour Sensor"
rectangle at (0,24)-(29,55): alarm colour if .ISenColourYellow
rectangle at (28,24)-(57,55): alarm colour if .ISenColourBlue
rectangle at (55,24)-(84,55): alarm colour if .ISenColourRed
rectangle at (82,24)-(111,55): alarm colour if .ISenColourGreen
*)

(* Visualisation Components/VC_Graph_Counters
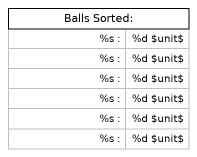
embedded screen at (0,20)-(181,41): VC_Var_Int
rectangle at (0,0)-(181,21): text "Balls Sorted:"
embedded screen at (0,40)-(181,61): VC_Var_Int
embedded screen at (0,60)-(181,81): VC_Var_Int
embedded screen at (0,80)-(181,101): VC_Var_Int
embedded screen at (0,120)-(181,141): VC_Var_Int
embedded screen at (0,100)-(181,121): VC_Var_Int
*)

(* Visualisation Components/VC_GRAPH_LIFT
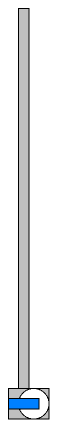
rectangle at (0,380)-(41,411): y offset -1 * PRG_HMI.iLiftPos
ellipse at (10,380)-(41,411): invisible if NOT .PRG_HMI.bBall_InLift; y offset -1 * PRG_HMI.iLiftPos
rectangle at (0,390)-(31,401): invisible if NOT .OEjector; y offset -1 * PRG_HMI.iLiftPos
1 more shapes without text or variables
*)

(* Visualisation Components/VC_GRAPH_SORTER
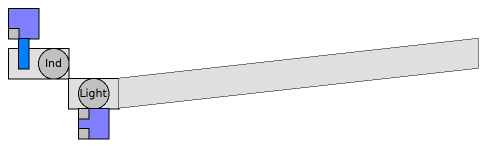
rectangle at (60,70)-(111,101): y offset -1 * PRG_HMI.iSorterLiftPos
rectangle at (10,30)-(21,61): invisible if .OSorterGate
ellipse at (70,70)-(101,101): text "Light"; alarm colour if .ISensorOpt; y offset -1 * PRG_HMI.iSorterLiftPos
ellipse at (30,40)-(61,71): text "Ind"; alarm colour if .ISensorInd
rectangle at (70,100)-(81,111): alarm colour if .ISorterLiftUp
rectangle at (70,120)-(81,131): alarm colour if .ISorterLiftDown
rectangle at (0,20)-(11,31): alarm colour if .ISorterGateClosed
6 more shapes without text or variables
*)

(* Visualisation Visual Components/VC_PackMLStates
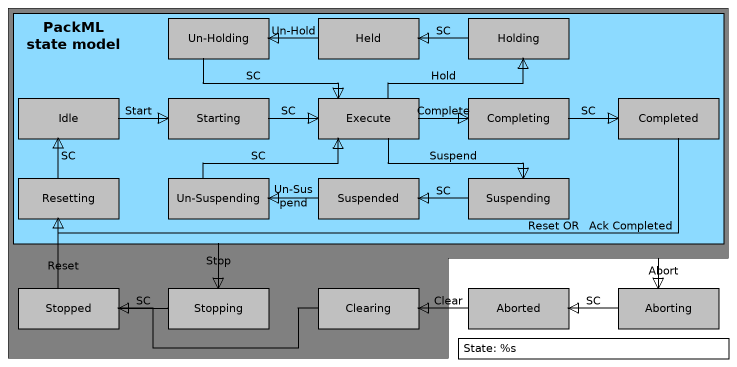
rounded rectangle at (160,280)-(261,321): text "Stopping"; alarm colour if $PackML$.eState = 4
rounded rectangle at (10,90)-(111,131): text "Idle"; alarm colour if $PackML$.eState = 6
rounded rectangle at (160,170)-(261,211): text "Un-Suspending"; alarm colour if $PackML$.eState = 11
rounded rectangle at (610,280)-(711,321): text "Aborting"; alarm colour if $PackML$.eState = 0
rounded rectangle at (460,280)-(561,321): text "Aborted"; alarm colour if $PackML$.eState = 1
rectangle at (450,330)-(721,351): text "State: %s"; shows .fbStateModel.eState
rounded rectangle at (310,280)-(411,321): text "Clearing"; alarm colour if $PackML$.eState = 2
rounded rectangle at (10,280)-(111,321): text "Stopped"; alarm colour if $PackML$.eState = 3
rounded rectangle at (10,170)-(111,211): text "Resetting"; alarm colour if $PackML$.eState = 5
rounded rectangle at (160,90)-(261,131): text "Starting"; alarm colour if $PackML$.eState = 7
rounded rectangle at (310,90)-(411,131): text "Execute"; alarm colour if $PackML$.eState = 8
rounded rectangle at (460,90)-(561,131): text "Completing"; alarm colour if $PackML$.eState = 15
rounded rectangle at (610,90)-(711,131): text "Completed"; alarm colour if $PackML$.eState = 16
rounded rectangle at (310,170)-(411,211): text "Suspended"; alarm colour if $PackML$.eState = 10
rounded rectangle at (460,170)-(561,211): text "Suspending"; alarm colour if $PackML$.eState = 9
rounded rectangle at (460,10)-(561,51): text "Holding"; alarm colour if $PackML$.eState = 12
rounded rectangle at (310,10)-(411,51): text "Held"; alarm colour if $PackML$.eState = 13
rounded rectangle at (160,10)-(261,51): text "Un-Holding"; alarm colour if $PackML$.eState = 14
polyline at (645,250)-(655,280): alarm colour if $PackML$.bAbort
rectangle at (635,255)-(676,271): text "Abort"; alarm colour if $PackML$.bAbort
polyline at (205,235)-(215,280): alarm colour if $PackML$.bStop
rectangle at (190,245)-(231,261): text "Stop"; alarm colour if $PackML$.bStop
polyline at (195,130)-(335,170): alarm colour if $PackML$.bSC
rectangle at (235,140)-(266,156): text "SC"; alarm colour if $PackML$.bSC
polyline at (195,50)-(335,90): alarm colour if $PackML$.bSC
polyline at (380,50)-(520,90): alarm colour if $PackML$.bHold
rectangle at (420,60)-(451,76): text "Hold"; alarm colour if $PackML$.bHold
polyline at (560,295)-(610,305): alarm colour if $PackML$.bSC
polyline at (45,210)-(55,280): alarm colour if $PackML$.bReset
polyline at (110,105)-(160,115): alarm colour if $PackML$.bStart
polyline at (110,295)-(310,340): alarm colour if $PackML$.bSC
rectangle at (230,60)-(261,76): text "SC"; alarm colour if $PackML$.bSC
polyline at (380,130)-(520,170): alarm colour if $PackML$.bSuspend
rectangle at (415,140)-(476,156): text "Suspend"; alarm colour if $PackML$.bSuspend
rectangle at (120,285)-(151,301): text "SC"; alarm colour if $PackML$.bSC
rectangle at (570,285)-(601,301): text "SC"; alarm colour if $PackML$.bSC
polyline at (410,295)-(460,305): alarm colour if $PackML$.bClear
rectangle at (420,285)-(461,301): text "Clear"; alarm colour if $PackML$.bClear
polyline at (260,105)-(310,115): alarm colour if $PackML$.bSC
rectangle at (265,95)-(296,111): text "SC"; alarm colour if $PackML$.bSC
rectangle at (110,95)-(151,111): text "Start"; alarm colour if $PackML$.bStart
rectangle at (35,250)-(76,266): text "Reset"; alarm colour if $PackML$.bReset
polyline at (410,185)-(460,195): alarm colour if $PackML$.bSC
rectangle at (420,175)-(451,191): text "SC"; alarm colour if $PackML$.bSC
polyline at (410,25)-(460,35): alarm colour if $PackML$.bSC
rectangle at (420,15)-(451,31): text "SC"; alarm colour if $PackML$.bSC
polyline at (260,185)-(310,195): alarm colour if $PackML$.bUn_Suspend
rectangle at (260,170)-(311,206): text "Un-Sus / pend"; alarm colour if $PackML$.bUn_Suspend
polyline at (260,25)-(310,35): alarm colour if $PackML$.bUn_Hold
rectangle at (260,15)-(311,31): text "Un-Hold"; alarm colour if $PackML$.bUn_Hold
polyline at (410,105)-(460,115): alarm colour if $PackML$.bComplete
rectangle at (410,95)-(461,111): text "Complete"; alarm colour if $PackML$.bComplete
polyline at (560,105)-(610,115): alarm colour if $PackML$.bSC
rectangle at (565,95)-(596,111): text "SC"; alarm colour if $PackML$.bSC
polyline at (45,130)-(55,170): alarm colour if $PackML$.bSC
rectangle at (45,140)-(76,156): text "SC"; alarm colour if $PackML$.bSC
polyline at (50,130)-(670,225): alarm colour if $PackML$.bReset OR $PackML$.Ack_Completed
rectangle at (515,210)-(576,226): text "Reset OR"; alarm colour if $PackML$.bReset
rectangle at (575,210)-(671,226): text "Ack Completed"; alarm colour if $PackML$.bAck_Completed
rectangle at (10,10)-(121,51): text "PackML / state model"
2 more shapes without text or variables
*)

(* Visualisation Simulator/MachineComponents/VC_PANEL_BATCHCONTROL
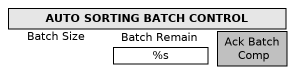
rectangle at (0,-3)-(278,18): text "AUTO SORTING BATCH CONTROL"
rectangle at (104,19)-(199,34): text "Batch Remain"
rectangle at (105,36)-(200,53): text "%s"; shows .iBatchRemaining
rectangle at (6,18)-(90,33): text "Batch Size"
rounded rectangle at (209,20)-(279,55): text "Ack Batch / Comp"; alarm colour if PRG_Sorting.bBatchComplete; taps .bHMI_BtnAck
1 elements of other kinds (tables, trends, ...) not read
*)

(* Visualisation Simulator/MachineComponents/VC_PANEL_MACHINECONTROL
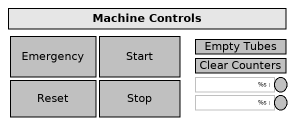
rounded rectangle at (2,28)-(88,69): text "Emergency"; alarm colour if NOT .IEmergencyClear
rounded rectangle at (91,28)-(172,69): text "Start"; alarm colour if .bHMI_BtnStartLight; taps .bHMI_BtnStart
rounded rectangle at (2,72)-(88,109): text "Reset"; taps bHMI_BtnReset
rounded rectangle at (91,72)-(172,109): text "Stop"; alarm colour if .bHMI_BtnStopLight; taps .bHMI_BtnStop
rectangle at (0,0)-(278,21): text "Machine Controls"
rounded rectangle at (187,31)-(278,46): text "Empty Tubes"; taps PRG_HMI.bBtnEmptyPipes
rounded rectangle at (187,50)-(278,65): text "Clear Counters"; taps PRG_HMI.bBtnResetCounters
embedded screen at (187,69)-(279,84): VC_BOOLEANSTATUS
embedded screen at (187,87)-(279,102): VC_BOOLEANSTATUS
1 more shapes without text or variables
*)

(* Visualisation Simulator/MachineComponents/VC_PANEL_MODESELECTOR
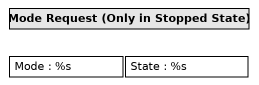
rectangle at (0,0)-(240,21): text "Mode Request (Only in Stopped State)"
rectangle at (0,48)-(114,69): text "Mode : %s"; shows .fbStateModel.eMode
rectangle at (116,48)-(239,69): text "State : %s"; shows .fbStateModel.eState
3 elements of other kinds (tables, trends, ...) not read
*)

(* Visualisation Simulator/MachineComponents/VC_PANEL_PROCMODESELECT
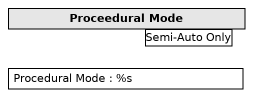
rectangle at (0,0)-(237,21): text "Proceedural Mode"
rectangle at (0,60)-(235,81): text "Procedural Mode : %s"; shows .fbStateModel.eMode
rectangle at (137,21)-(224,38): text "Semi-Auto Only"
3 elements of other kinds (tables, trends, ...) not read
*)

(* Visualisation Components/VC_PIPE
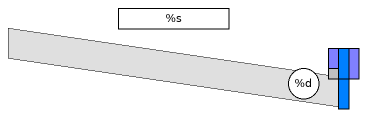
rectangle at (330,70)-(361,101): invisible if NOT .IPressureApplied
rectangle at (340,100)-(351,131): invisible if NOT $FB$.I_GateClosed  OR NOT .IPressureApplied; tooltip Output cmd to open gate
rectangle at (330,90)-(341,101): alarm colour if $FB$.I_GateClosed; tooltip Gate is closed input
ellipse at (290,90)-(321,121): text "%d"; shows $FB$.iBallCount
rectangle at (120,30)-(231,51): text "%s"; shows $FB$.str_PipeName
rectangle at (340,70)-(351,101): tooltip Output cmd to open gate
2 more shapes without text or variables
*)

(* Visualisation Simulator/Components/VC_sensor
rectangle at (0,0)-(11,11): alarm colour if $VAR$
*)

(* Visualisation Components/VC_Var_Int
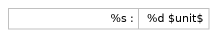
rectangle at (0,0)-(131,21): text "%s :"; shows $Name$
rectangle at (130,0)-(201,21): text "%d $unit$"; shows $VAR$
*)
